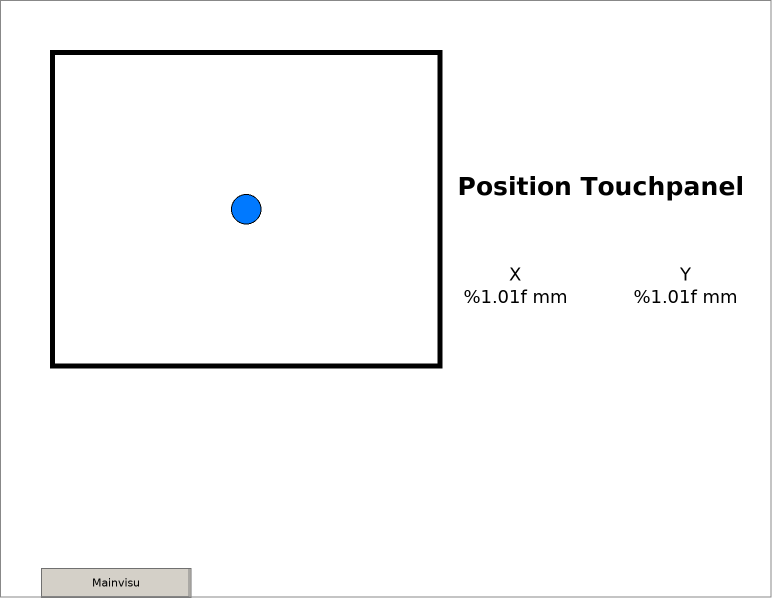
VISUALIZATION Touch  // 772x598
    Rectangle (50,50 392x318)
    Ellipse (231,194 30x30), invisible if: NOT Touchpanel.bContactAvailable
        p3560616238: -Touchpanel.touch_scale_x.rX_mm
        p2738717112: Touchpanel.touch_scale_y.rX_mm
    Rectangle (600,260 171x51), "Y %1.01f mm", text variable: Touchpanel.touch_scale_y.rX_mm
    Rectangle (430,260 171x51), "X %1.01f mm", text variable: Touchpanel.touch_scale_x.rX_mm
    Label (430,156 342x60), "Position Touchpanel"
    Button (41,568 150x30), "Mainvisu"
        OnMouseDown: change screen: Mainvisu
END_VISUALIZATION

(* stored: Version 1.1.0.1, ProductVersion 3.1.4024.12
   Visu Touch: Id {af132e0e-c432-4516-b716-945794d96eeb} *)
